{attribute 'qualified_only'}
{attribute 'strict'}
TYPE E_PISTON_STATE :
(
	uninit:=0,
	ready,
	opening,
	opened,
	closing,
	closed,
	error,
	busy
);
END_TYPE

(* stored: Version 1.1.0.1, ProductVersion 3.1.4024.12
   DUT E_PISTON_STATE: Id {0e8efeed-2681-40cd-bfae-c5b4d1cd92b4} *)
